// TIA Portal V19 export
VAR_GLOBAL   // PLC tag table "Standard-Variablentabelle"
   start AT %I0.0 : Bool;
   motor AT %Q0.0 : Bool;
   stop AT %I0.1 : Bool;
   mem AT %M0.2 : Bool;
END_VAR
